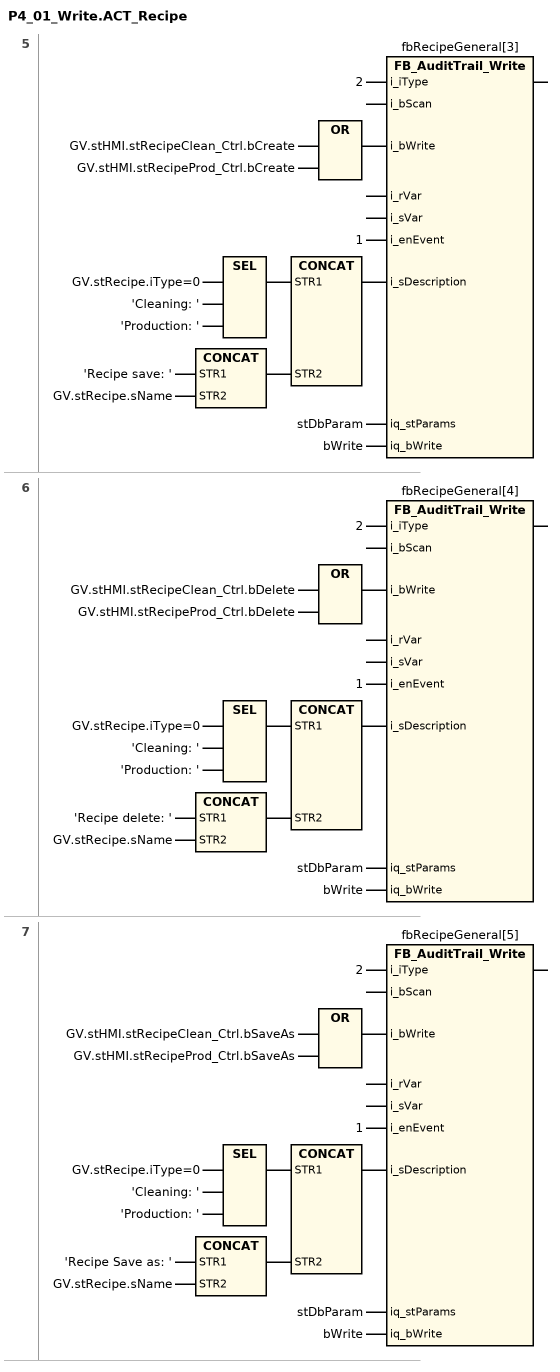
// NETWORK 5
fbRecipeGeneral[3](
    i_iType := 2,
    i_bWrite := GV.stHMI.stRecipeClean_Ctrl.bCreate OR GV.stHMI.stRecipeProd_Ctrl.bCreate,
    i_enEvent := 1,
    i_sDescription := CONCAT(STR1 := SEL(GV.stRecipe.iType=0, 'Cleaning: ', 'Production: '), STR2 := CONCAT(STR1 := 'Recipe save: ', STR2 := GV.stRecipe.sName)),
    iq_stParams := stDbParam,
    iq_bWrite := bWrite); // FB_AuditTrail_Write

// NETWORK 6
fbRecipeGeneral[4](
    i_iType := 2,
    i_bWrite := GV.stHMI.stRecipeClean_Ctrl.bDelete OR GV.stHMI.stRecipeProd_Ctrl.bDelete,
    i_enEvent := 1,
    i_sDescription := CONCAT(STR1 := SEL(GV.stRecipe.iType=0, 'Cleaning: ', 'Production: '), STR2 := CONCAT(STR1 := 'Recipe delete: ', STR2 := GV.stRecipe.sName)),
    iq_stParams := stDbParam,
    iq_bWrite := bWrite); // FB_AuditTrail_Write

// NETWORK 7
fbRecipeGeneral[5](
    i_iType := 2,
    i_bWrite := GV.stHMI.stRecipeClean_Ctrl.bSaveAs OR GV.stHMI.stRecipeProd_Ctrl.bSaveAs,
    i_enEvent := 1,
    i_sDescription := CONCAT(STR1 := SEL(GV.stRecipe.iType=0, 'Cleaning: ', 'Production: '), STR2 := CONCAT(STR1 := 'Recipe Save as: ', STR2 := GV.stRecipe.sName)),
    iq_stParams := stDbParam,
    iq_bWrite := bWrite); // FB_AuditTrail_Write

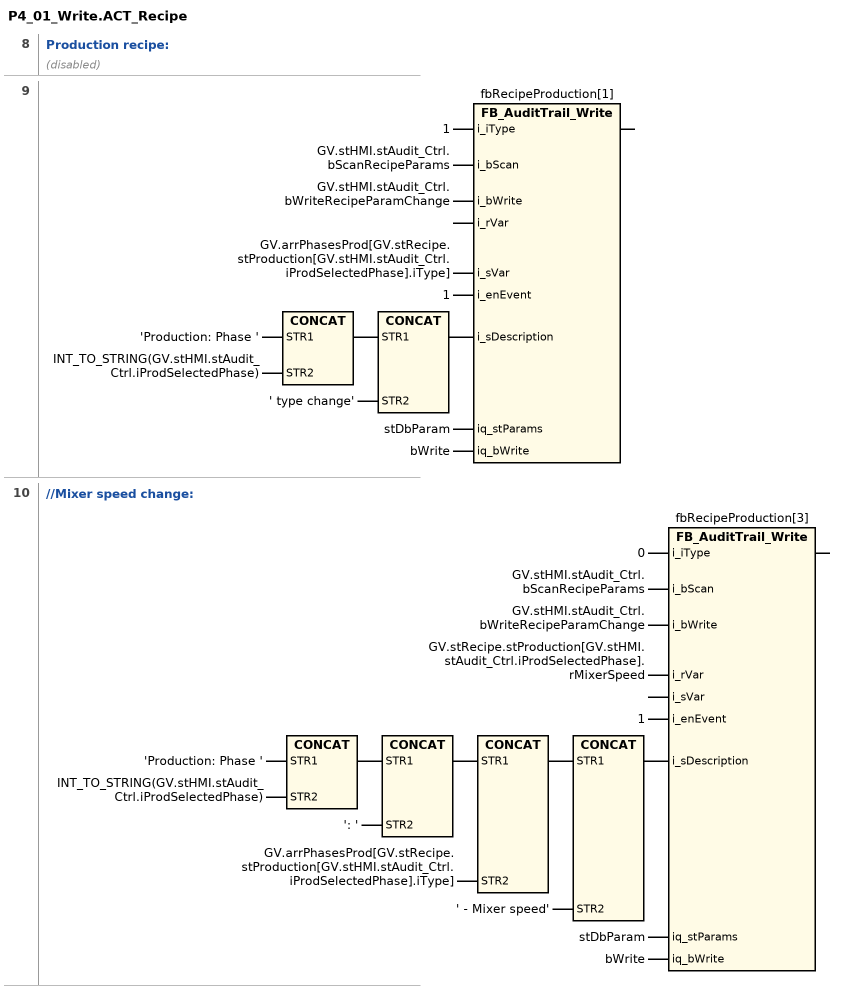
// NETWORK 8 (disabled)
// label: Production recipe

// NETWORK 9
fbRecipeProduction[1](
    i_iType := 1,
    i_bScan := GV.stHMI.stAudit_Ctrl.bScanRecipeParams,
    i_bWrite := GV.stHMI.stAudit_Ctrl.bWriteRecipeParamChange,
    i_sVar := GV.arrPhasesProd[GV.stRecipe.stProduction[GV.stHMI.stAudit_Ctrl.iProdSelectedPhase].iType],
    i_enEvent := 1,
    i_sDescription := CONCAT(STR1 := CONCAT(STR1 := 'Production: Phase ', STR2 := INT_TO_STRING(GV.stHMI.stAudit_Ctrl.iProdSelectedPhase)), STR2 := ' type change'),
    iq_stParams := stDbParam,
    iq_bWrite := bWrite); // FB_AuditTrail_Write

// NETWORK 10
// label: //Mixer speed change
fbRecipeProduction[3](
    i_iType := 0,
    i_bScan := GV.stHMI.stAudit_Ctrl.bScanRecipeParams,
    i_bWrite := GV.stHMI.stAudit_Ctrl.bWriteRecipeParamChange,
    i_rVar := GV.stRecipe.stProduction[GV.stHMI.stAudit_Ctrl.iProdSelectedPhase].rMixerSpeed,
    i_enEvent := 1,
    i_sDescription := CONCAT(STR1 := CONCAT(STR1 := CONCAT(STR1 := CONCAT(STR1 := 'Production: Phase ', STR2 := INT_TO_STRING(GV.stHMI.stAudit_Ctrl.iProdSelectedPhase)), STR2 := ': '), STR2 := GV.arrPhasesProd[GV.stRecipe.stProduction[GV.stHMI.stAudit_Ctrl.iProdSelectedPhase].iType]), STR2 := ' - Mixer speed'),
    iq_stParams := stDbParam,
    iq_bWrite := bWrite); // FB_AuditTrail_Write

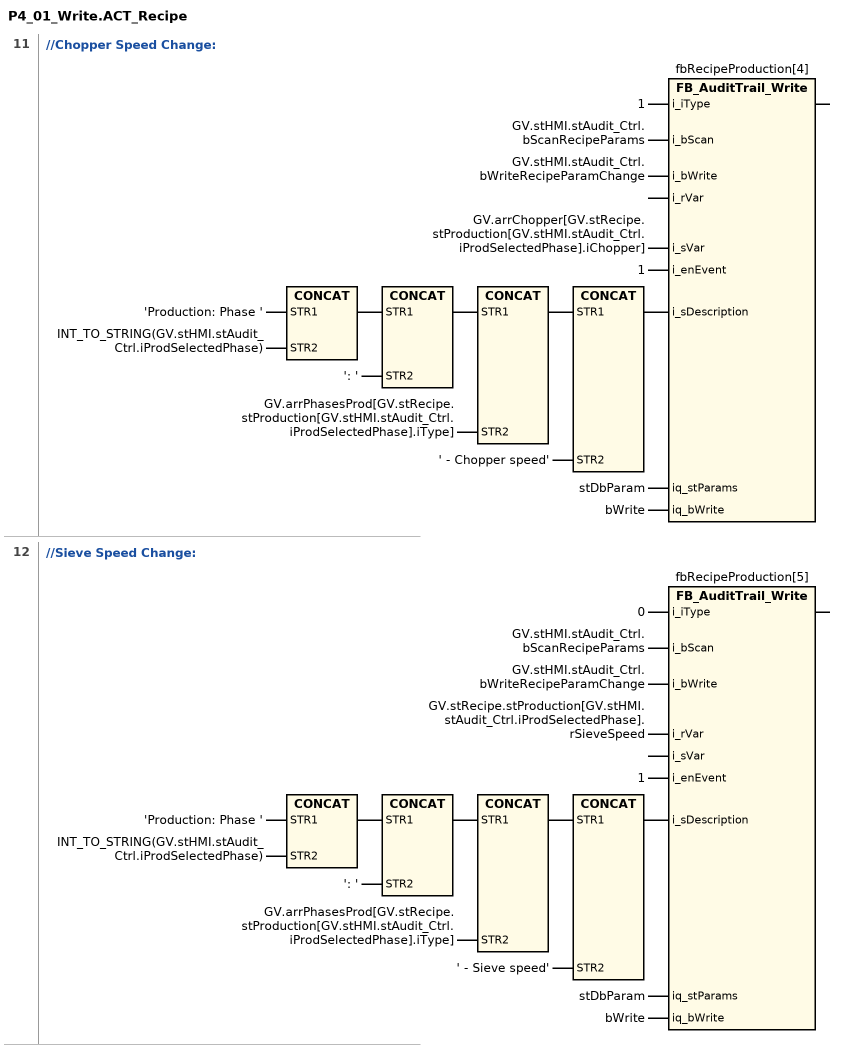
// NETWORK 11
// label: //Chopper Speed Change
fbRecipeProduction[4](
    i_iType := 1,
    i_bScan := GV.stHMI.stAudit_Ctrl.bScanRecipeParams,
    i_bWrite := GV.stHMI.stAudit_Ctrl.bWriteRecipeParamChange,
    i_sVar := GV.arrChopper[GV.stRecipe.stProduction[GV.stHMI.stAudit_Ctrl.iProdSelectedPhase].iChopper],
    i_enEvent := 1,
    i_sDescription := CONCAT(STR1 := CONCAT(STR1 := CONCAT(STR1 := CONCAT(STR1 := 'Production: Phase ', STR2 := INT_TO_STRING(GV.stHMI.stAudit_Ctrl.iProdSelectedPhase)), STR2 := ': '), STR2 := GV.arrPhasesProd[GV.stRecipe.stProduction[GV.stHMI.stAudit_Ctrl.iProdSelectedPhase].iType]), STR2 := ' - Chopper speed'),
    iq_stParams := stDbParam,
    iq_bWrite := bWrite); // FB_AuditTrail_Write

// NETWORK 12
// label: //Sieve Speed Change
fbRecipeProduction[5](
    i_iType := 0,
    i_bScan := GV.stHMI.stAudit_Ctrl.bScanRecipeParams,
    i_bWrite := GV.stHMI.stAudit_Ctrl.bWriteRecipeParamChange,
    i_rVar := GV.stRecipe.stProduction[GV.stHMI.stAudit_Ctrl.iProdSelectedPhase].rSieveSpeed,
    i_enEvent := 1,
    i_sDescription := CONCAT(STR1 := CONCAT(STR1 := CONCAT(STR1 := CONCAT(STR1 := 'Production: Phase ', STR2 := INT_TO_STRING(GV.stHMI.stAudit_Ctrl.iProdSelectedPhase)), STR2 := ': '), STR2 := GV.arrPhasesProd[GV.stRecipe.stProduction[GV.stHMI.stAudit_Ctrl.iProdSelectedPhase].iType]), STR2 := ' - Sieve speed'),
    iq_stParams := stDbParam,
    iq_bWrite := bWrite); // FB_AuditTrail_Write

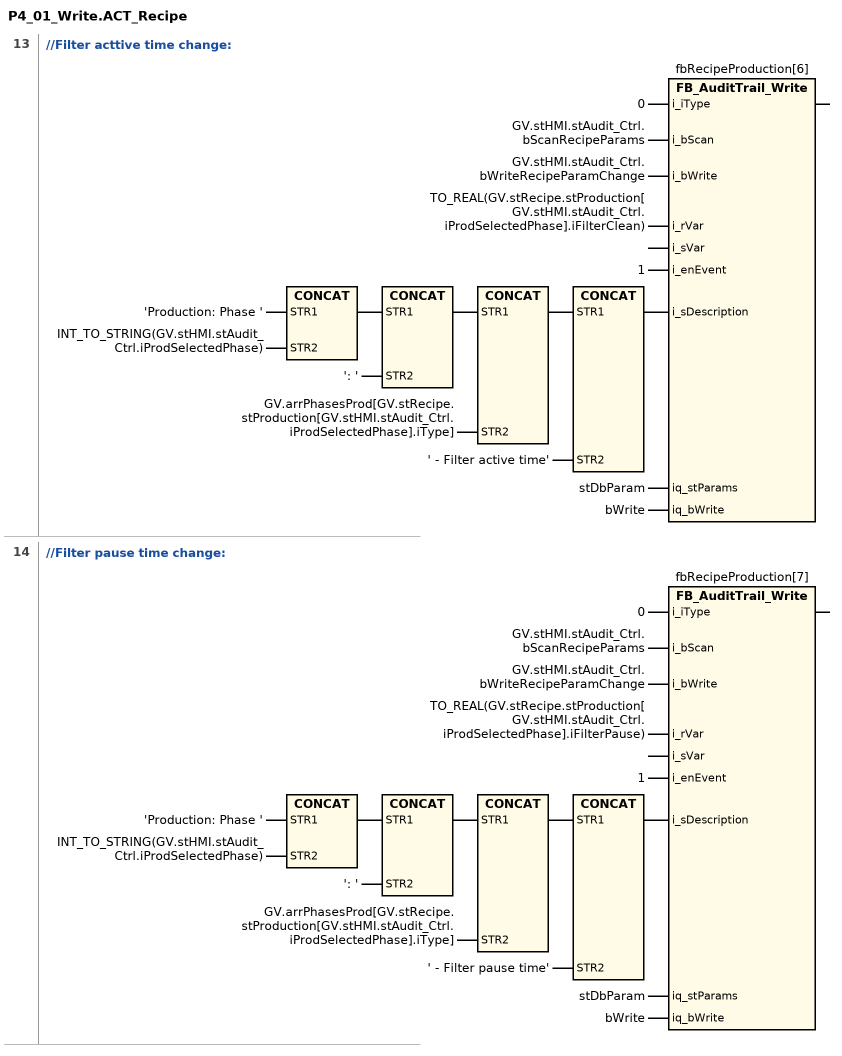
// NETWORK 13
// label: //Filter acttive time change
fbRecipeProduction[6](
    i_iType := 0,
    i_bScan := GV.stHMI.stAudit_Ctrl.bScanRecipeParams,
    i_bWrite := GV.stHMI.stAudit_Ctrl.bWriteRecipeParamChange,
    i_rVar := TO_REAL(GV.stRecipe.stProduction[GV.stHMI.stAudit_Ctrl.iProdSelectedPhase].iFilterClean),
    i_enEvent := 1,
    i_sDescription := CONCAT(STR1 := CONCAT(STR1 := CONCAT(STR1 := CONCAT(STR1 := 'Production: Phase ', STR2 := INT_TO_STRING(GV.stHMI.stAudit_Ctrl.iProdSelectedPhase)), STR2 := ': '), STR2 := GV.arrPhasesProd[GV.stRecipe.stProduction[GV.stHMI.stAudit_Ctrl.iProdSelectedPhase].iType]), STR2 := ' - Filter active time'),
    iq_stParams := stDbParam,
    iq_bWrite := bWrite); // FB_AuditTrail_Write

// NETWORK 14
// label: //Filter pause time change
fbRecipeProduction[7](
    i_iType := 0,
    i_bScan := GV.stHMI.stAudit_Ctrl.bScanRecipeParams,
    i_bWrite := GV.stHMI.stAudit_Ctrl.bWriteRecipeParamChange,
    i_rVar := TO_REAL(GV.stRecipe.stProduction[GV.stHMI.stAudit_Ctrl.iProdSelectedPhase].iFilterPause),
    i_enEvent := 1,
    i_sDescription := CONCAT(STR1 := CONCAT(STR1 := CONCAT(STR1 := CONCAT(STR1 := 'Production: Phase ', STR2 := INT_TO_STRING(GV.stHMI.stAudit_Ctrl.iProdSelectedPhase)), STR2 := ': '), STR2 := GV.arrPhasesProd[GV.stRecipe.stProduction[GV.stHMI.stAudit_Ctrl.iProdSelectedPhase].iType]), STR2 := ' - Filter pause time'),
    iq_stParams := stDbParam,
    iq_bWrite := bWrite); // FB_AuditTrail_Write

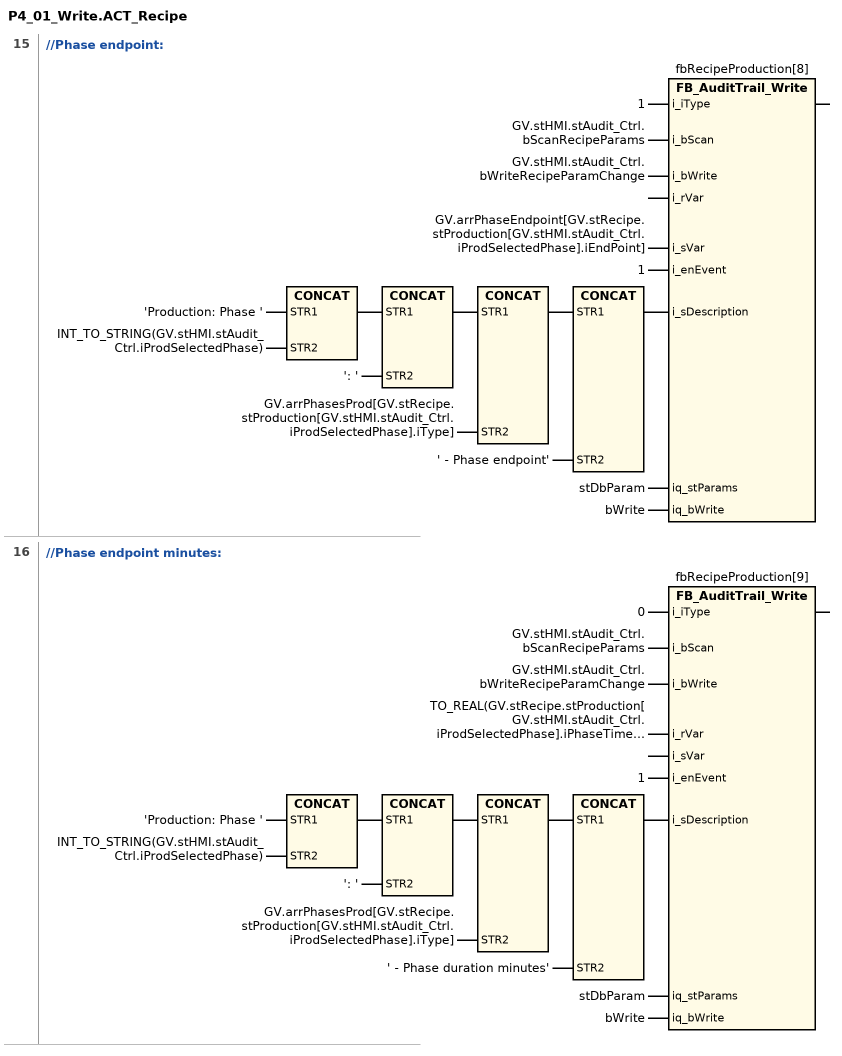
// NETWORK 15
// label: //Phase endpoint
fbRecipeProduction[8](
    i_iType := 1,
    i_bScan := GV.stHMI.stAudit_Ctrl.bScanRecipeParams,
    i_bWrite := GV.stHMI.stAudit_Ctrl.bWriteRecipeParamChange,
    i_sVar := GV.arrPhaseEndpoint[GV.stRecipe.stProduction[GV.stHMI.stAudit_Ctrl.iProdSelectedPhase].iEndPoint],
    i_enEvent := 1,
    i_sDescription := CONCAT(STR1 := CONCAT(STR1 := CONCAT(STR1 := CONCAT(STR1 := 'Production: Phase ', STR2 := INT_TO_STRING(GV.stHMI.stAudit_Ctrl.iProdSelectedPhase)), STR2 := ': '), STR2 := GV.arrPhasesProd[GV.stRecipe.stProduction[GV.stHMI.stAudit_Ctrl.iProdSelectedPhase].iType]), STR2 := ' - Phase endpoint'),
    iq_stParams := stDbParam,
    iq_bWrite := bWrite); // FB_AuditTrail_Write

// NETWORK 16
// label: //Phase endpoint minutes
fbRecipeProduction[9](
    i_iType := 0,
    i_bScan := GV.stHMI.stAudit_Ctrl.bScanRecipeParams,
    i_bWrite := GV.stHMI.stAudit_Ctrl.bWriteRecipeParamChange,
    i_rVar := TO_REAL(GV.stRecipe.stProduction[GV.stHMI.stAudit_Ctrl.iProdSelectedPhase].iPhaseTime.mins),
    i_enEvent := 1,
    i_sDescription := CONCAT(STR1 := CONCAT(STR1 := CONCAT(STR1 := CONCAT(STR1 := 'Production: Phase ', STR2 := INT_TO_STRING(GV.stHMI.stAudit_Ctrl.iProdSelectedPhase)), STR2 := ': '), STR2 := GV.arrPhasesProd[GV.stRecipe.stProduction[GV.stHMI.stAudit_Ctrl.iProdSelectedPhase].iType]), STR2 := ' - Phase duration minutes'),
    iq_stParams := stDbParam,
    iq_bWrite := bWrite); // FB_AuditTrail_Write

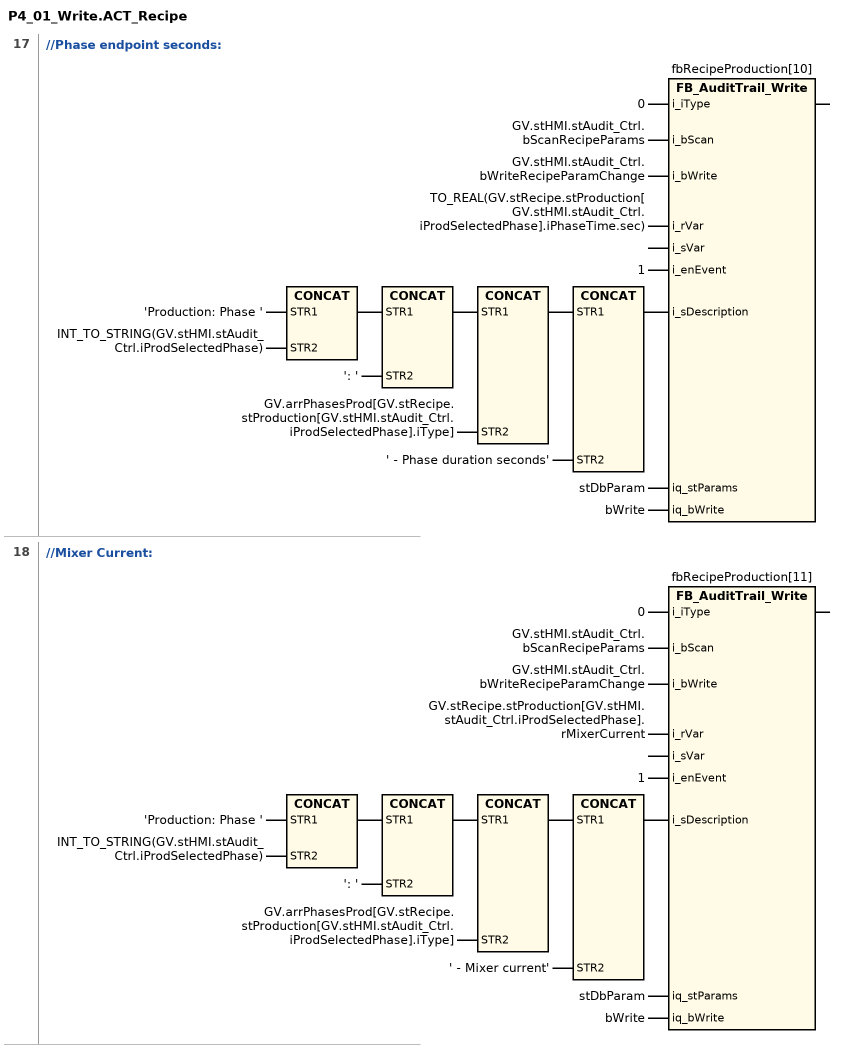
// NETWORK 17
// label: //Phase endpoint seconds
fbRecipeProduction[10](
    i_iType := 0,
    i_bScan := GV.stHMI.stAudit_Ctrl.bScanRecipeParams,
    i_bWrite := GV.stHMI.stAudit_Ctrl.bWriteRecipeParamChange,
    i_rVar := TO_REAL(GV.stRecipe.stProduction[GV.stHMI.stAudit_Ctrl.iProdSelectedPhase].iPhaseTime.sec),
    i_enEvent := 1,
    i_sDescription := CONCAT(STR1 := CONCAT(STR1 := CONCAT(STR1 := CONCAT(STR1 := 'Production: Phase ', STR2 := INT_TO_STRING(GV.stHMI.stAudit_Ctrl.iProdSelectedPhase)), STR2 := ': '), STR2 := GV.arrPhasesProd[GV.stRecipe.stProduction[GV.stHMI.stAudit_Ctrl.iProdSelectedPhase].iType]), STR2 := ' - Phase duration seconds'),
    iq_stParams := stDbParam,
    iq_bWrite := bWrite); // FB_AuditTrail_Write

// NETWORK 18
// label: //Mixer Current
fbRecipeProduction[11](
    i_iType := 0,
    i_bScan := GV.stHMI.stAudit_Ctrl.bScanRecipeParams,
    i_bWrite := GV.stHMI.stAudit_Ctrl.bWriteRecipeParamChange,
    i_rVar := GV.stRecipe.stProduction[GV.stHMI.stAudit_Ctrl.iProdSelectedPhase].rMixerCurrent,
    i_enEvent := 1,
    i_sDescription := CONCAT(STR1 := CONCAT(STR1 := CONCAT(STR1 := CONCAT(STR1 := 'Production: Phase ', STR2 := INT_TO_STRING(GV.stHMI.stAudit_Ctrl.iProdSelectedPhase)), STR2 := ': '), STR2 := GV.arrPhasesProd[GV.stRecipe.stProduction[GV.stHMI.stAudit_Ctrl.iProdSelectedPhase].iType]), STR2 := ' - Mixer current'),
    iq_stParams := stDbParam,
    iq_bWrite := bWrite); // FB_AuditTrail_Write

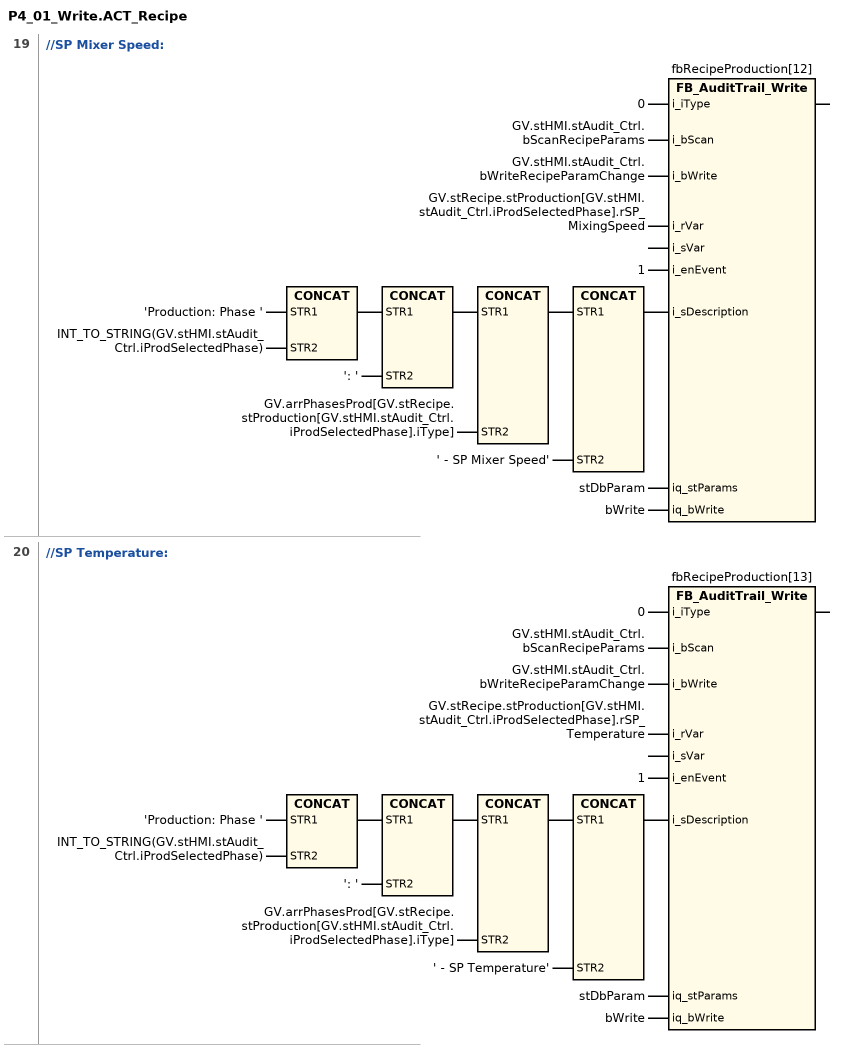
// NETWORK 19
// label: //SP Mixer Speed
fbRecipeProduction[12](
    i_iType := 0,
    i_bScan := GV.stHMI.stAudit_Ctrl.bScanRecipeParams,
    i_bWrite := GV.stHMI.stAudit_Ctrl.bWriteRecipeParamChange,
    i_rVar := GV.stRecipe.stProduction[GV.stHMI.stAudit_Ctrl.iProdSelectedPhase].rSP_MixingSpeed,
    i_enEvent := 1,
    i_sDescription := CONCAT(STR1 := CONCAT(STR1 := CONCAT(STR1 := CONCAT(STR1 := 'Production: Phase ', STR2 := INT_TO_STRING(GV.stHMI.stAudit_Ctrl.iProdSelectedPhase)), STR2 := ': '), STR2 := GV.arrPhasesProd[GV.stRecipe.stProduction[GV.stHMI.stAudit_Ctrl.iProdSelectedPhase].iType]), STR2 := ' - SP Mixer Speed'),
    iq_stParams := stDbParam,
    iq_bWrite := bWrite); // FB_AuditTrail_Write

// NETWORK 20
// label: //SP Temperature
fbRecipeProduction[13](
    i_iType := 0,
    i_bScan := GV.stHMI.stAudit_Ctrl.bScanRecipeParams,
    i_bWrite := GV.stHMI.stAudit_Ctrl.bWriteRecipeParamChange,
    i_rVar := GV.stRecipe.stProduction[GV.stHMI.stAudit_Ctrl.iProdSelectedPhase].rSP_Temperature,
    i_enEvent := 1,
    i_sDescription := CONCAT(STR1 := CONCAT(STR1 := CONCAT(STR1 := CONCAT(STR1 := 'Production: Phase ', STR2 := INT_TO_STRING(GV.stHMI.stAudit_Ctrl.iProdSelectedPhase)), STR2 := ': '), STR2 := GV.arrPhasesProd[GV.stRecipe.stProduction[GV.stHMI.stAudit_Ctrl.iProdSelectedPhase].iType]), STR2 := ' - SP Temperature'),
    iq_stParams := stDbParam,
    iq_bWrite := bWrite); // FB_AuditTrail_Write

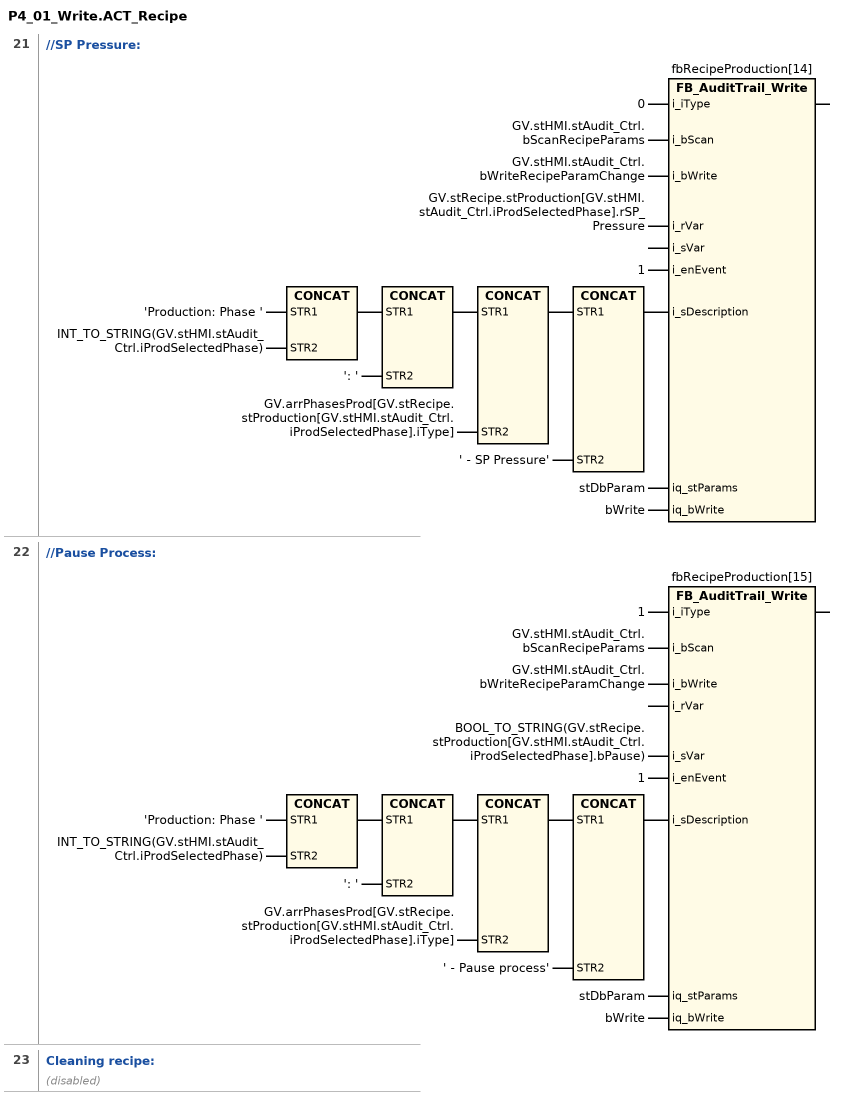
// NETWORK 21
// label: //SP Pressure
fbRecipeProduction[14](
    i_iType := 0,
    i_bScan := GV.stHMI.stAudit_Ctrl.bScanRecipeParams,
    i_bWrite := GV.stHMI.stAudit_Ctrl.bWriteRecipeParamChange,
    i_rVar := GV.stRecipe.stProduction[GV.stHMI.stAudit_Ctrl.iProdSelectedPhase].rSP_Pressure,
    i_enEvent := 1,
    i_sDescription := CONCAT(STR1 := CONCAT(STR1 := CONCAT(STR1 := CONCAT(STR1 := 'Production: Phase ', STR2 := INT_TO_STRING(GV.stHMI.stAudit_Ctrl.iProdSelectedPhase)), STR2 := ': '), STR2 := GV.arrPhasesProd[GV.stRecipe.stProduction[GV.stHMI.stAudit_Ctrl.iProdSelectedPhase].iType]), STR2 := ' - SP Pressure'),
    iq_stParams := stDbParam,
    iq_bWrite := bWrite); // FB_AuditTrail_Write

// NETWORK 22
// label: //Pause Process
fbRecipeProduction[15](
    i_iType := 1,
    i_bScan := GV.stHMI.stAudit_Ctrl.bScanRecipeParams,
    i_bWrite := GV.stHMI.stAudit_Ctrl.bWriteRecipeParamChange,
    i_sVar := BOOL_TO_STRING(GV.stRecipe.stProduction[GV.stHMI.stAudit_Ctrl.iProdSelectedPhase].bPause),
    i_enEvent := 1,
    i_sDescription := CONCAT(STR1 := CONCAT(STR1 := CONCAT(STR1 := CONCAT(STR1 := 'Production: Phase ', STR2 := INT_TO_STRING(GV.stHMI.stAudit_Ctrl.iProdSelectedPhase)), STR2 := ': '), STR2 := GV.arrPhasesProd[GV.stRecipe.stProduction[GV.stHMI.stAudit_Ctrl.iProdSelectedPhase].iType]), STR2 := ' - Pause process'),
    iq_stParams := stDbParam,
    iq_bWrite := bWrite); // FB_AuditTrail_Write

// NETWORK 23 (disabled)
// label: Cleaning recipe

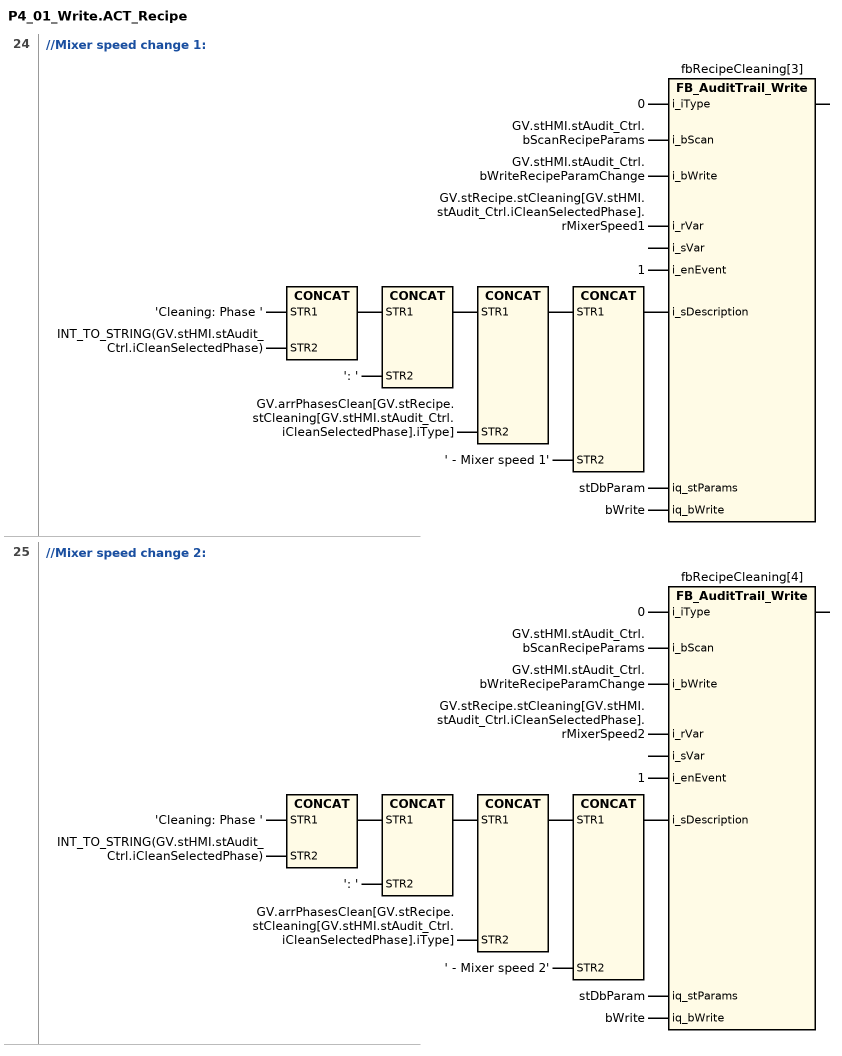
// NETWORK 24
// label: //Mixer speed change 1
fbRecipeCleaning[3](
    i_iType := 0,
    i_bScan := GV.stHMI.stAudit_Ctrl.bScanRecipeParams,
    i_bWrite := GV.stHMI.stAudit_Ctrl.bWriteRecipeParamChange,
    i_rVar := GV.stRecipe.stCleaning[GV.stHMI.stAudit_Ctrl.iCleanSelectedPhase].rMixerSpeed1,
    i_enEvent := 1,
    i_sDescription := CONCAT(STR1 := CONCAT(STR1 := CONCAT(STR1 := CONCAT(STR1 := 'Cleaning: Phase ', STR2 := INT_TO_STRING(GV.stHMI.stAudit_Ctrl.iCleanSelectedPhase)), STR2 := ': '), STR2 := GV.arrPhasesClean[GV.stRecipe.stCleaning[GV.stHMI.stAudit_Ctrl.iCleanSelectedPhase].iType]), STR2 := ' - Mixer speed 1'),
    iq_stParams := stDbParam,
    iq_bWrite := bWrite); // FB_AuditTrail_Write

// NETWORK 25
// label: //Mixer speed change 2
fbRecipeCleaning[4](
    i_iType := 0,
    i_bScan := GV.stHMI.stAudit_Ctrl.bScanRecipeParams,
    i_bWrite := GV.stHMI.stAudit_Ctrl.bWriteRecipeParamChange,
    i_rVar := GV.stRecipe.stCleaning[GV.stHMI.stAudit_Ctrl.iCleanSelectedPhase].rMixerSpeed2,
    i_enEvent := 1,
    i_sDescription := CONCAT(STR1 := CONCAT(STR1 := CONCAT(STR1 := CONCAT(STR1 := 'Cleaning: Phase ', STR2 := INT_TO_STRING(GV.stHMI.stAudit_Ctrl.iCleanSelectedPhase)), STR2 := ': '), STR2 := GV.arrPhasesClean[GV.stRecipe.stCleaning[GV.stHMI.stAudit_Ctrl.iCleanSelectedPhase].iType]), STR2 := ' - Mixer speed 2'),
    iq_stParams := stDbParam,
    iq_bWrite := bWrite); // FB_AuditTrail_Write

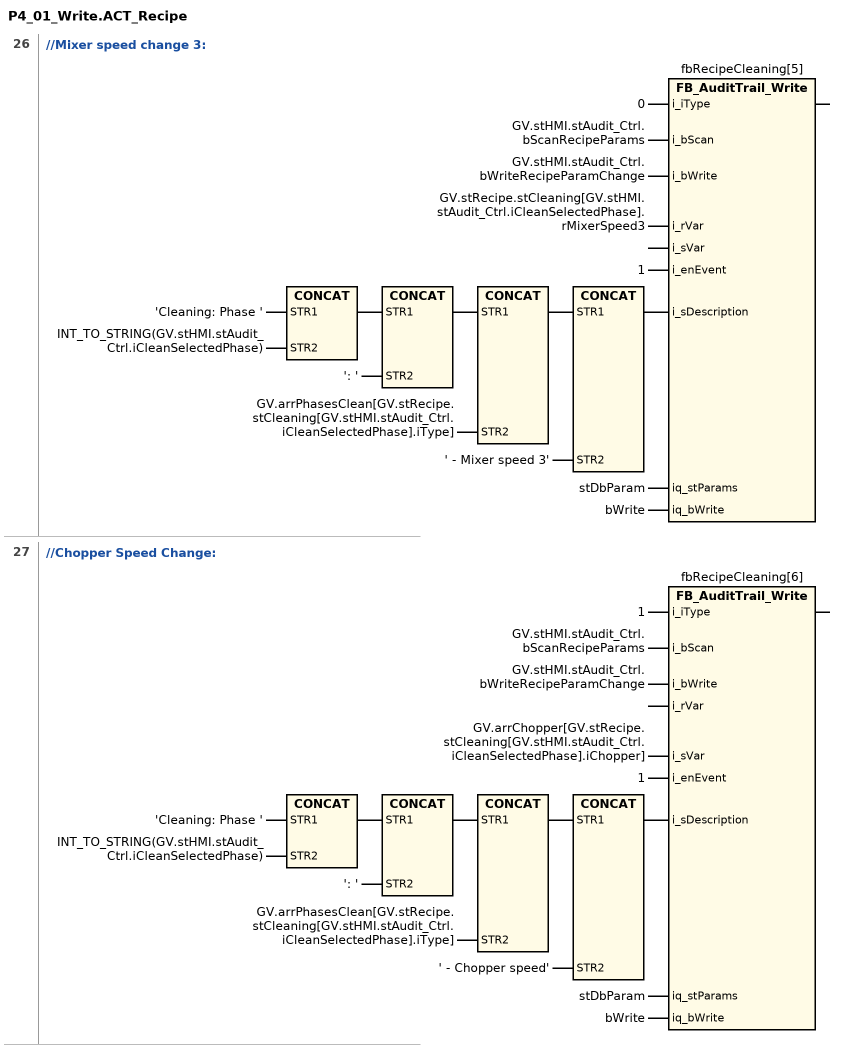
// NETWORK 26
// label: //Mixer speed change 3
fbRecipeCleaning[5](
    i_iType := 0,
    i_bScan := GV.stHMI.stAudit_Ctrl.bScanRecipeParams,
    i_bWrite := GV.stHMI.stAudit_Ctrl.bWriteRecipeParamChange,
    i_rVar := GV.stRecipe.stCleaning[GV.stHMI.stAudit_Ctrl.iCleanSelectedPhase].rMixerSpeed3,
    i_enEvent := 1,
    i_sDescription := CONCAT(STR1 := CONCAT(STR1 := CONCAT(STR1 := CONCAT(STR1 := 'Cleaning: Phase ', STR2 := INT_TO_STRING(GV.stHMI.stAudit_Ctrl.iCleanSelectedPhase)), STR2 := ': '), STR2 := GV.arrPhasesClean[GV.stRecipe.stCleaning[GV.stHMI.stAudit_Ctrl.iCleanSelectedPhase].iType]), STR2 := ' - Mixer speed 3'),
    iq_stParams := stDbParam,
    iq_bWrite := bWrite); // FB_AuditTrail_Write

// NETWORK 27
// label: //Chopper Speed Change
fbRecipeCleaning[6](
    i_iType := 1,
    i_bScan := GV.stHMI.stAudit_Ctrl.bScanRecipeParams,
    i_bWrite := GV.stHMI.stAudit_Ctrl.bWriteRecipeParamChange,
    i_sVar := GV.arrChopper[GV.stRecipe.stCleaning[GV.stHMI.stAudit_Ctrl.iCleanSelectedPhase].iChopper],
    i_enEvent := 1,
    i_sDescription := CONCAT(STR1 := CONCAT(STR1 := CONCAT(STR1 := CONCAT(STR1 := 'Cleaning: Phase ', STR2 := INT_TO_STRING(GV.stHMI.stAudit_Ctrl.iCleanSelectedPhase)), STR2 := ': '), STR2 := GV.arrPhasesClean[GV.stRecipe.stCleaning[GV.stHMI.stAudit_Ctrl.iCleanSelectedPhase].iType]), STR2 := ' - Chopper speed'),
    iq_stParams := stDbParam,
    iq_bWrite := bWrite); // FB_AuditTrail_Write

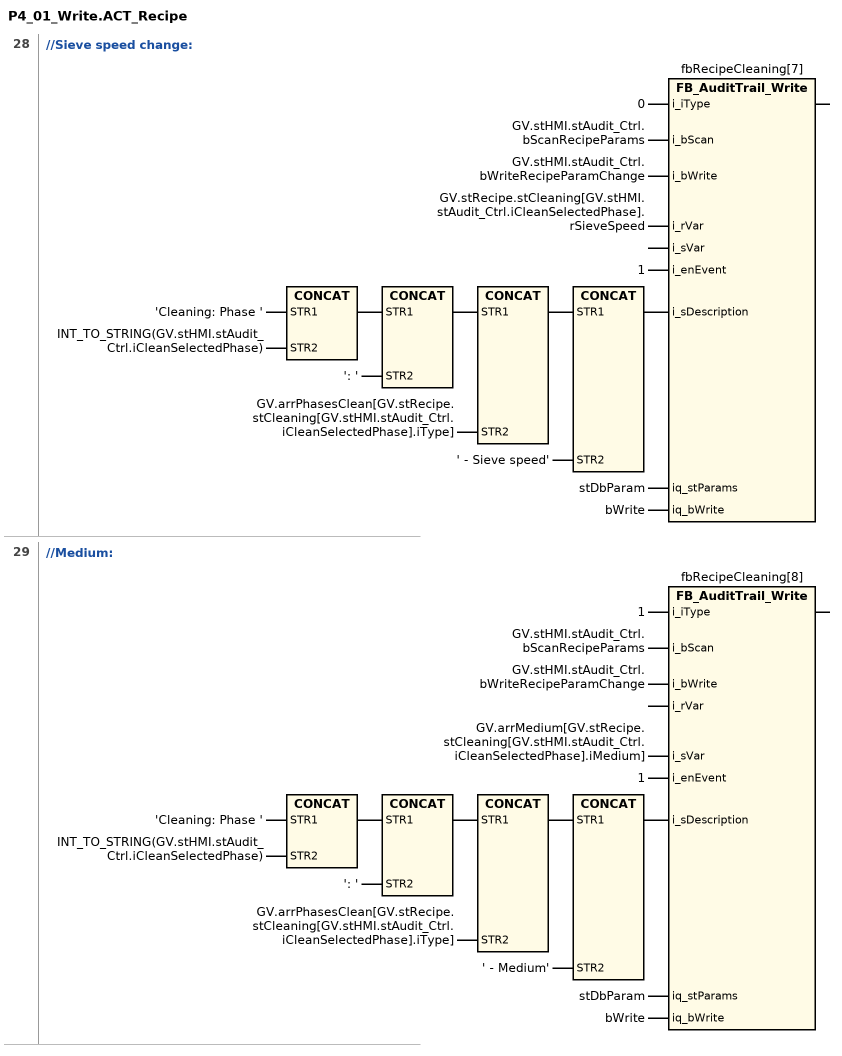
// NETWORK 28
// label: //Sieve speed change
fbRecipeCleaning[7](
    i_iType := 0,
    i_bScan := GV.stHMI.stAudit_Ctrl.bScanRecipeParams,
    i_bWrite := GV.stHMI.stAudit_Ctrl.bWriteRecipeParamChange,
    i_rVar := GV.stRecipe.stCleaning[GV.stHMI.stAudit_Ctrl.iCleanSelectedPhase].rSieveSpeed,
    i_enEvent := 1,
    i_sDescription := CONCAT(STR1 := CONCAT(STR1 := CONCAT(STR1 := CONCAT(STR1 := 'Cleaning: Phase ', STR2 := INT_TO_STRING(GV.stHMI.stAudit_Ctrl.iCleanSelectedPhase)), STR2 := ': '), STR2 := GV.arrPhasesClean[GV.stRecipe.stCleaning[GV.stHMI.stAudit_Ctrl.iCleanSelectedPhase].iType]), STR2 := ' - Sieve speed'),
    iq_stParams := stDbParam,
    iq_bWrite := bWrite); // FB_AuditTrail_Write

// NETWORK 29
// label: //Medium
fbRecipeCleaning[8](
    i_iType := 1,
    i_bScan := GV.stHMI.stAudit_Ctrl.bScanRecipeParams,
    i_bWrite := GV.stHMI.stAudit_Ctrl.bWriteRecipeParamChange,
    i_sVar := GV.arrMedium[GV.stRecipe.stCleaning[GV.stHMI.stAudit_Ctrl.iCleanSelectedPhase].iMedium],
    i_enEvent := 1,
    i_sDescription := CONCAT(STR1 := CONCAT(STR1 := CONCAT(STR1 := CONCAT(STR1 := 'Cleaning: Phase ', STR2 := INT_TO_STRING(GV.stHMI.stAudit_Ctrl.iCleanSelectedPhase)), STR2 := ': '), STR2 := GV.arrPhasesClean[GV.stRecipe.stCleaning[GV.stHMI.stAudit_Ctrl.iCleanSelectedPhase].iType]), STR2 := ' - Medium'),
    iq_stParams := stDbParam,
    iq_bWrite := bWrite); // FB_AuditTrail_Write

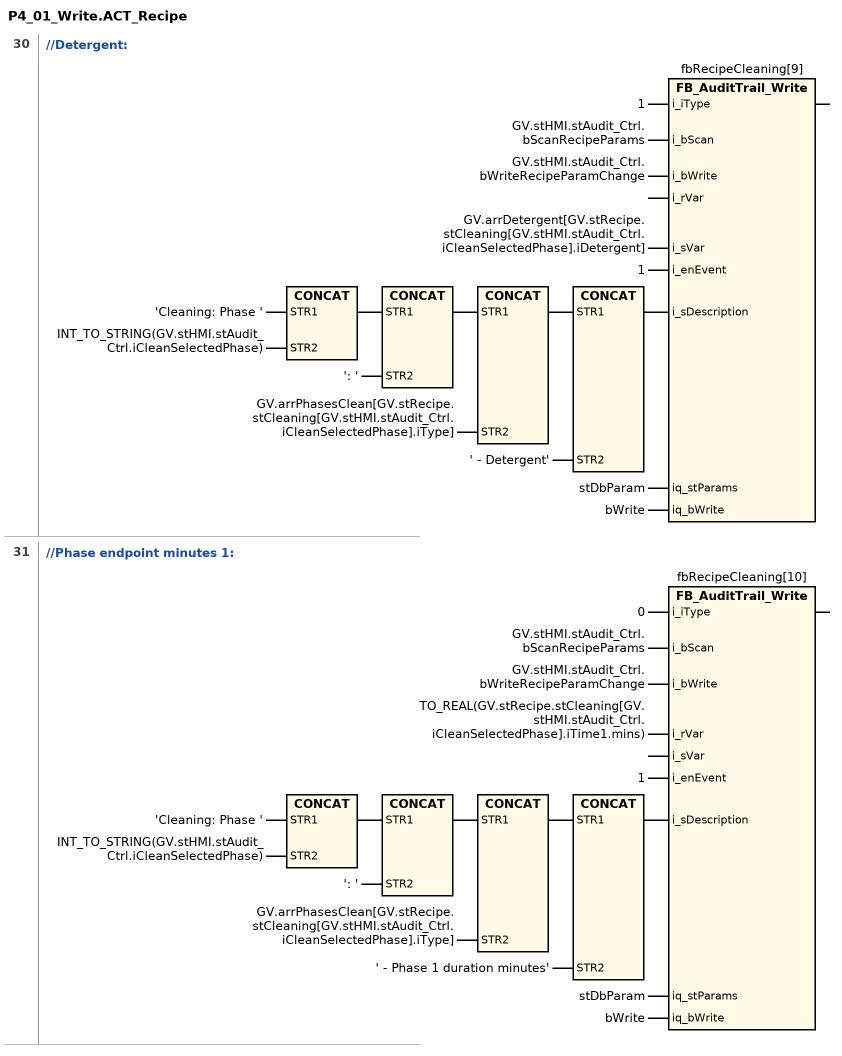
// NETWORK 30
// label: //Detergent
fbRecipeCleaning[9](
    i_iType := 1,
    i_bScan := GV.stHMI.stAudit_Ctrl.bScanRecipeParams,
    i_bWrite := GV.stHMI.stAudit_Ctrl.bWriteRecipeParamChange,
    i_sVar := GV.arrDetergent[GV.stRecipe.stCleaning[GV.stHMI.stAudit_Ctrl.iCleanSelectedPhase].iDetergent],
    i_enEvent := 1,
    i_sDescription := CONCAT(STR1 := CONCAT(STR1 := CONCAT(STR1 := CONCAT(STR1 := 'Cleaning: Phase ', STR2 := INT_TO_STRING(GV.stHMI.stAudit_Ctrl.iCleanSelectedPhase)), STR2 := ': '), STR2 := GV.arrPhasesClean[GV.stRecipe.stCleaning[GV.stHMI.stAudit_Ctrl.iCleanSelectedPhase].iType]), STR2 := ' - Detergent'),
    iq_stParams := stDbParam,
    iq_bWrite := bWrite); // FB_AuditTrail_Write

// NETWORK 31
// label: //Phase endpoint minutes 1
fbRecipeCleaning[10](
    i_iType := 0,
    i_bScan := GV.stHMI.stAudit_Ctrl.bScanRecipeParams,
    i_bWrite := GV.stHMI.stAudit_Ctrl.bWriteRecipeParamChange,
    i_rVar := TO_REAL(GV.stRecipe.stCleaning[GV.stHMI.stAudit_Ctrl.iCleanSelectedPhase].iTime1.mins),
    i_enEvent := 1,
    i_sDescription := CONCAT(STR1 := CONCAT(STR1 := CONCAT(STR1 := CONCAT(STR1 := 'Cleaning: Phase ', STR2 := INT_TO_STRING(GV.stHMI.stAudit_Ctrl.iCleanSelectedPhase)), STR2 := ': '), STR2 := GV.arrPhasesClean[GV.stRecipe.stCleaning[GV.stHMI.stAudit_Ctrl.iCleanSelectedPhase].iType]), STR2 := ' - Phase 1 duration minutes'),
    iq_stParams := stDbParam,
    iq_bWrite := bWrite); // FB_AuditTrail_Write

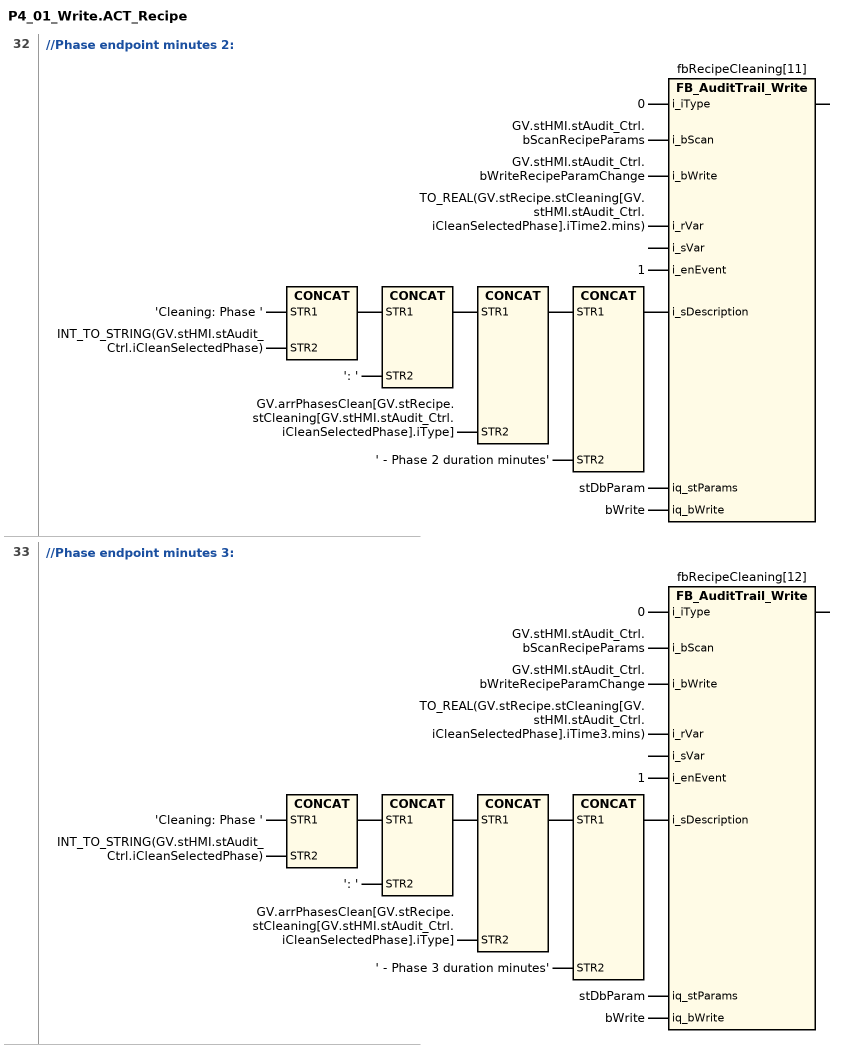
// NETWORK 32
// label: //Phase endpoint minutes 2
fbRecipeCleaning[11](
    i_iType := 0,
    i_bScan := GV.stHMI.stAudit_Ctrl.bScanRecipeParams,
    i_bWrite := GV.stHMI.stAudit_Ctrl.bWriteRecipeParamChange,
    i_rVar := TO_REAL(GV.stRecipe.stCleaning[GV.stHMI.stAudit_Ctrl.iCleanSelectedPhase].iTime2.mins),
    i_enEvent := 1,
    i_sDescription := CONCAT(STR1 := CONCAT(STR1 := CONCAT(STR1 := CONCAT(STR1 := 'Cleaning: Phase ', STR2 := INT_TO_STRING(GV.stHMI.stAudit_Ctrl.iCleanSelectedPhase)), STR2 := ': '), STR2 := GV.arrPhasesClean[GV.stRecipe.stCleaning[GV.stHMI.stAudit_Ctrl.iCleanSelectedPhase].iType]), STR2 := ' - Phase 2 duration minutes'),
    iq_stParams := stDbParam,
    iq_bWrite := bWrite); // FB_AuditTrail_Write

// NETWORK 33
// label: //Phase endpoint minutes 3
fbRecipeCleaning[12](
    i_iType := 0,
    i_bScan := GV.stHMI.stAudit_Ctrl.bScanRecipeParams,
    i_bWrite := GV.stHMI.stAudit_Ctrl.bWriteRecipeParamChange,
    i_rVar := TO_REAL(GV.stRecipe.stCleaning[GV.stHMI.stAudit_Ctrl.iCleanSelectedPhase].iTime3.mins),
    i_enEvent := 1,
    i_sDescription := CONCAT(STR1 := CONCAT(STR1 := CONCAT(STR1 := CONCAT(STR1 := 'Cleaning: Phase ', STR2 := INT_TO_STRING(GV.stHMI.stAudit_Ctrl.iCleanSelectedPhase)), STR2 := ': '), STR2 := GV.arrPhasesClean[GV.stRecipe.stCleaning[GV.stHMI.stAudit_Ctrl.iCleanSelectedPhase].iType]), STR2 := ' - Phase 3 duration minutes'),
    iq_stParams := stDbParam,
    iq_bWrite := bWrite); // FB_AuditTrail_Write

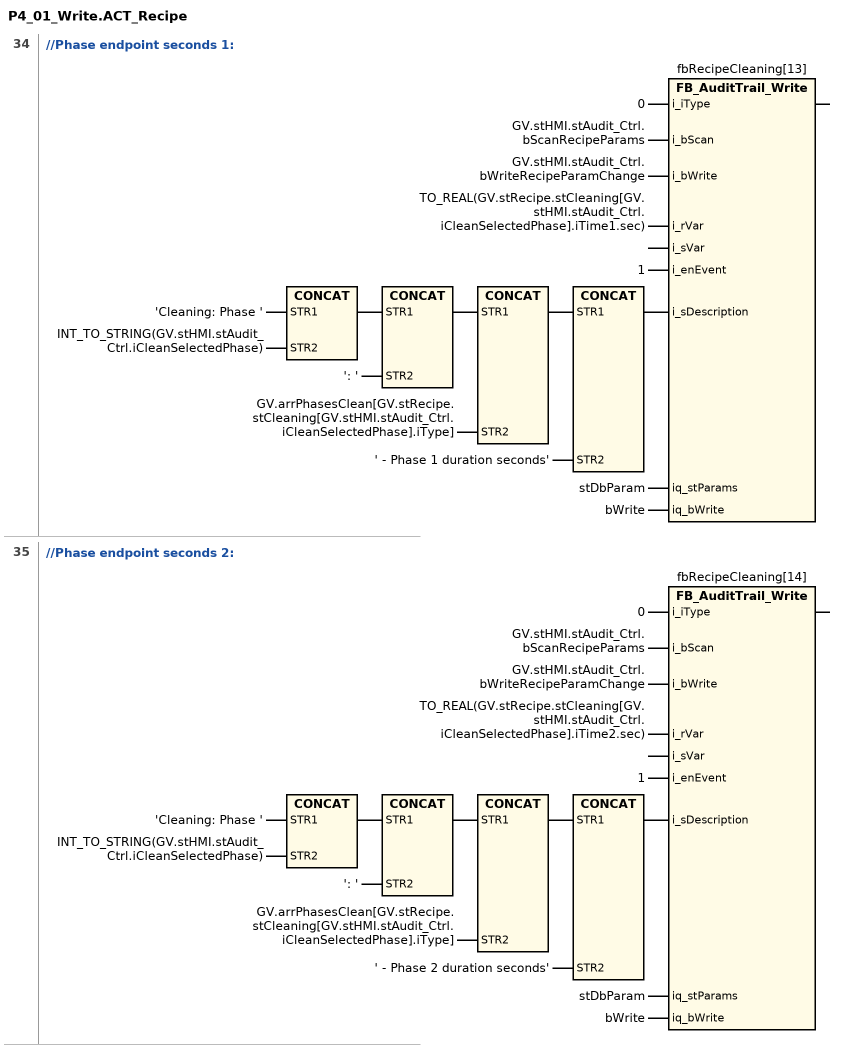
// NETWORK 34
// label: //Phase endpoint seconds 1
fbRecipeCleaning[13](
    i_iType := 0,
    i_bScan := GV.stHMI.stAudit_Ctrl.bScanRecipeParams,
    i_bWrite := GV.stHMI.stAudit_Ctrl.bWriteRecipeParamChange,
    i_rVar := TO_REAL(GV.stRecipe.stCleaning[GV.stHMI.stAudit_Ctrl.iCleanSelectedPhase].iTime1.sec),
    i_enEvent := 1,
    i_sDescription := CONCAT(STR1 := CONCAT(STR1 := CONCAT(STR1 := CONCAT(STR1 := 'Cleaning: Phase ', STR2 := INT_TO_STRING(GV.stHMI.stAudit_Ctrl.iCleanSelectedPhase)), STR2 := ': '), STR2 := GV.arrPhasesClean[GV.stRecipe.stCleaning[GV.stHMI.stAudit_Ctrl.iCleanSelectedPhase].iType]), STR2 := ' - Phase 1 duration seconds'),
    iq_stParams := stDbParam,
    iq_bWrite := bWrite); // FB_AuditTrail_Write

// NETWORK 35
// label: //Phase endpoint seconds 2
fbRecipeCleaning[14](
    i_iType := 0,
    i_bScan := GV.stHMI.stAudit_Ctrl.bScanRecipeParams,
    i_bWrite := GV.stHMI.stAudit_Ctrl.bWriteRecipeParamChange,
    i_rVar := TO_REAL(GV.stRecipe.stCleaning[GV.stHMI.stAudit_Ctrl.iCleanSelectedPhase].iTime2.sec),
    i_enEvent := 1,
    i_sDescription := CONCAT(STR1 := CONCAT(STR1 := CONCAT(STR1 := CONCAT(STR1 := 'Cleaning: Phase ', STR2 := INT_TO_STRING(GV.stHMI.stAudit_Ctrl.iCleanSelectedPhase)), STR2 := ': '), STR2 := GV.arrPhasesClean[GV.stRecipe.stCleaning[GV.stHMI.stAudit_Ctrl.iCleanSelectedPhase].iType]), STR2 := ' - Phase 2 duration seconds'),
    iq_stParams := stDbParam,
    iq_bWrite := bWrite); // FB_AuditTrail_Write

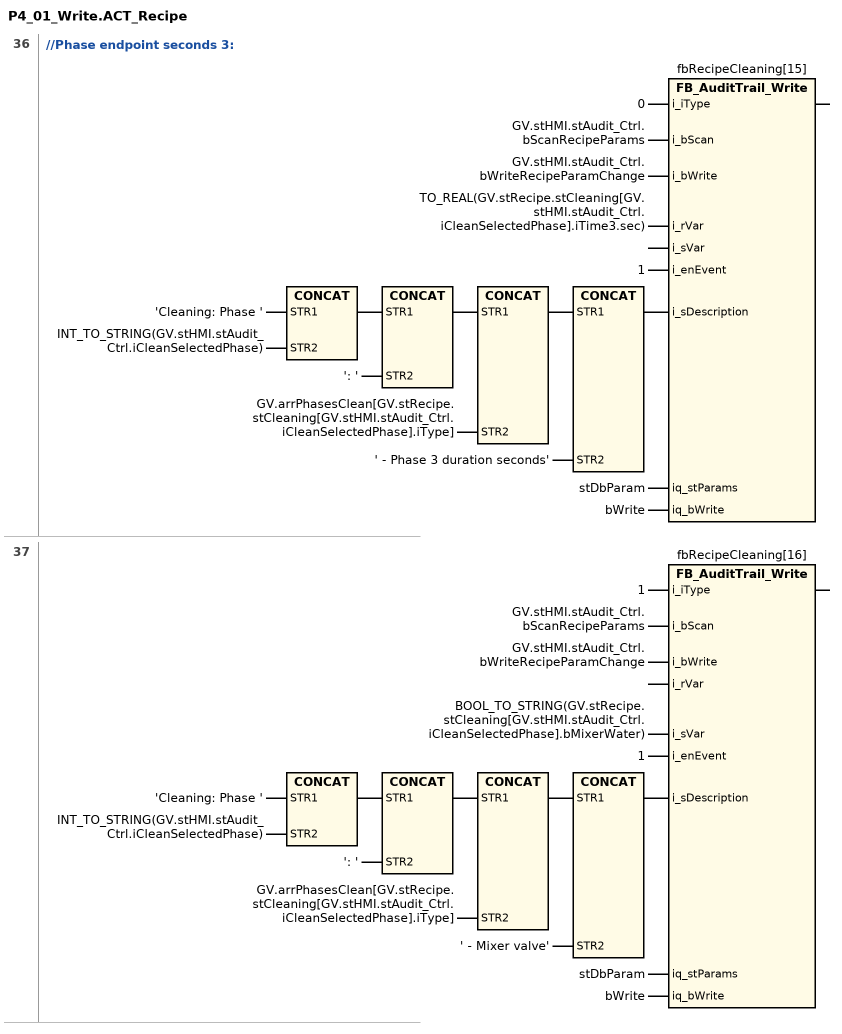
// NETWORK 36
// label: //Phase endpoint seconds 3
fbRecipeCleaning[15](
    i_iType := 0,
    i_bScan := GV.stHMI.stAudit_Ctrl.bScanRecipeParams,
    i_bWrite := GV.stHMI.stAudit_Ctrl.bWriteRecipeParamChange,
    i_rVar := TO_REAL(GV.stRecipe.stCleaning[GV.stHMI.stAudit_Ctrl.iCleanSelectedPhase].iTime3.sec),
    i_enEvent := 1,
    i_sDescription := CONCAT(STR1 := CONCAT(STR1 := CONCAT(STR1 := CONCAT(STR1 := 'Cleaning: Phase ', STR2 := INT_TO_STRING(GV.stHMI.stAudit_Ctrl.iCleanSelectedPhase)), STR2 := ': '), STR2 := GV.arrPhasesClean[GV.stRecipe.stCleaning[GV.stHMI.stAudit_Ctrl.iCleanSelectedPhase].iType]), STR2 := ' - Phase 3 duration seconds'),
    iq_stParams := stDbParam,
    iq_bWrite := bWrite); // FB_AuditTrail_Write

// NETWORK 37
fbRecipeCleaning[16](
    i_iType := 1,
    i_bScan := GV.stHMI.stAudit_Ctrl.bScanRecipeParams,
    i_bWrite := GV.stHMI.stAudit_Ctrl.bWriteRecipeParamChange,
    i_sVar := BOOL_TO_STRING(GV.stRecipe.stCleaning[GV.stHMI.stAudit_Ctrl.iCleanSelectedPhase].bMixerWater),
    i_enEvent := 1,
    i_sDescription := CONCAT(STR1 := CONCAT(STR1 := CONCAT(STR1 := CONCAT(STR1 := 'Cleaning: Phase ', STR2 := INT_TO_STRING(GV.stHMI.stAudit_Ctrl.iCleanSelectedPhase)), STR2 := ': '), STR2 := GV.arrPhasesClean[GV.stRecipe.stCleaning[GV.stHMI.stAudit_Ctrl.iCleanSelectedPhase].iType]), STR2 := ' - Mixer valve'),
    iq_stParams := stDbParam,
    iq_bWrite := bWrite); // FB_AuditTrail_Write

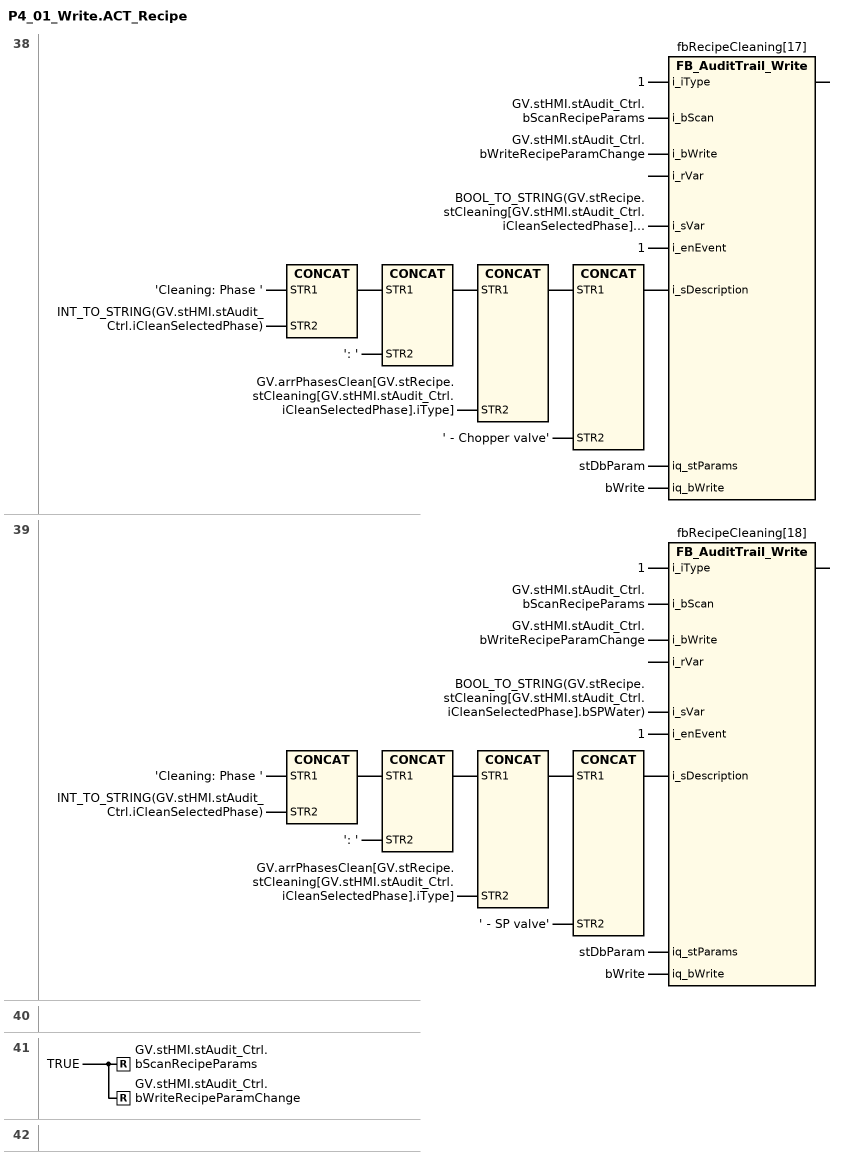
// NETWORK 38
fbRecipeCleaning[17](
    i_iType := 1,
    i_bScan := GV.stHMI.stAudit_Ctrl.bScanRecipeParams,
    i_bWrite := GV.stHMI.stAudit_Ctrl.bWriteRecipeParamChange,
    i_sVar := BOOL_TO_STRING(GV.stRecipe.stCleaning[GV.stHMI.stAudit_Ctrl.iCleanSelectedPhase].bChopperWater),
    i_enEvent := 1,
    i_sDescription := CONCAT(STR1 := CONCAT(STR1 := CONCAT(STR1 := CONCAT(STR1 := 'Cleaning: Phase ', STR2 := INT_TO_STRING(GV.stHMI.stAudit_Ctrl.iCleanSelectedPhase)), STR2 := ': '), STR2 := GV.arrPhasesClean[GV.stRecipe.stCleaning[GV.stHMI.stAudit_Ctrl.iCleanSelectedPhase].iType]), STR2 := ' - Chopper valve'),
    iq_stParams := stDbParam,
    iq_bWrite := bWrite); // FB_AuditTrail_Write

// NETWORK 39
fbRecipeCleaning[18](
    i_iType := 1,
    i_bScan := GV.stHMI.stAudit_Ctrl.bScanRecipeParams,
    i_bWrite := GV.stHMI.stAudit_Ctrl.bWriteRecipeParamChange,
    i_sVar := BOOL_TO_STRING(GV.stRecipe.stCleaning[GV.stHMI.stAudit_Ctrl.iCleanSelectedPhase].bSPWater),
    i_enEvent := 1,
    i_sDescription := CONCAT(STR1 := CONCAT(STR1 := CONCAT(STR1 := CONCAT(STR1 := 'Cleaning: Phase ', STR2 := INT_TO_STRING(GV.stHMI.stAudit_Ctrl.iCleanSelectedPhase)), STR2 := ': '), STR2 := GV.arrPhasesClean[GV.stRecipe.stCleaning[GV.stHMI.stAudit_Ctrl.iCleanSelectedPhase].iType]), STR2 := ' - SP valve'),
    iq_stParams := stDbParam,
    iq_bWrite := bWrite); // FB_AuditTrail_Write

// NETWORK 40

// NETWORK 41
GV.stHMI.stAudit_Ctrl.bScanRecipeParams R= TRUE;
GV.stHMI.stAudit_Ctrl.bWriteRecipeParamChange R= TRUE;

// NETWORK 42
END_ACTION

ACTION ACT_SP:
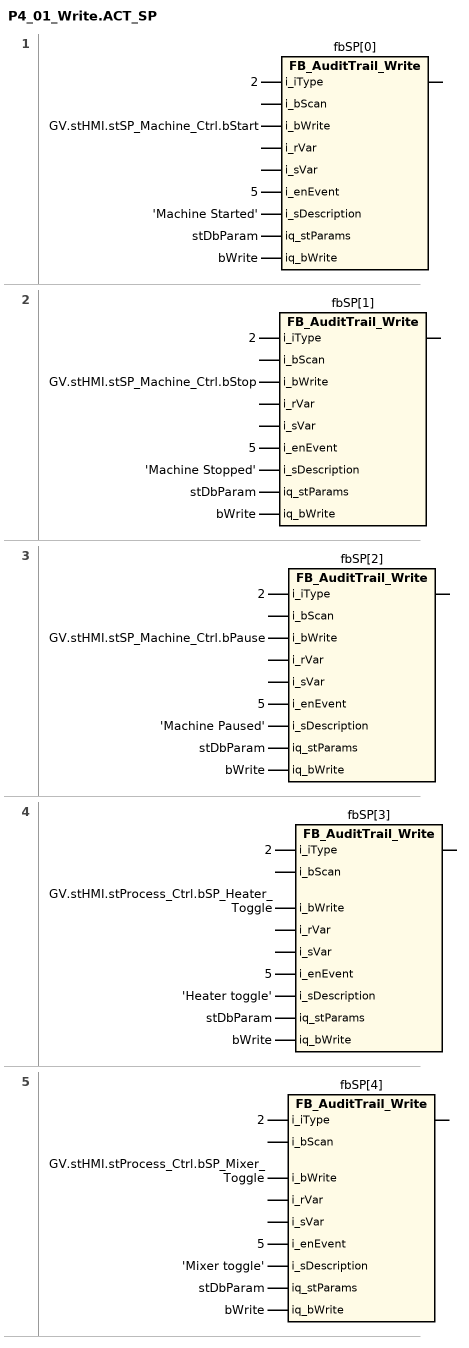
// NETWORK 1
fbSP[0](
    i_iType := 2,
    i_bWrite := GV.stHMI.stSP_Machine_Ctrl.bStart,
    i_enEvent := 5,
    i_sDescription := 'Machine Started',
    iq_stParams := stDbParam,
    iq_bWrite := bWrite); // FB_AuditTrail_Write

// NETWORK 2
fbSP[1](
    i_iType := 2,
    i_bWrite := GV.stHMI.stSP_Machine_Ctrl.bStop,
    i_enEvent := 5,
    i_sDescription := 'Machine Stopped',
    iq_stParams := stDbParam,
    iq_bWrite := bWrite); // FB_AuditTrail_Write

// NETWORK 3
fbSP[2](
    i_iType := 2,
    i_bWrite := GV.stHMI.stSP_Machine_Ctrl.bPause,
    i_enEvent := 5,
    i_sDescription := 'Machine Paused',
    iq_stParams := stDbParam,
    iq_bWrite := bWrite); // FB_AuditTrail_Write

// NETWORK 4
fbSP[3](
    i_iType := 2,
    i_bWrite := GV.stHMI.stProcess_Ctrl.bSP_Heater_Toggle,
    i_enEvent := 5,
    i_sDescription := 'Heater toggle',
    iq_stParams := stDbParam,
    iq_bWrite := bWrite); // FB_AuditTrail_Write

// NETWORK 5
fbSP[4](
    i_iType := 2,
    i_bWrite := GV.stHMI.stProcess_Ctrl.bSP_Mixer_Toggle,
    i_enEvent := 5,
    i_sDescription := 'Mixer toggle',
    iq_stParams := stDbParam,
    iq_bWrite := bWrite); // FB_AuditTrail_Write

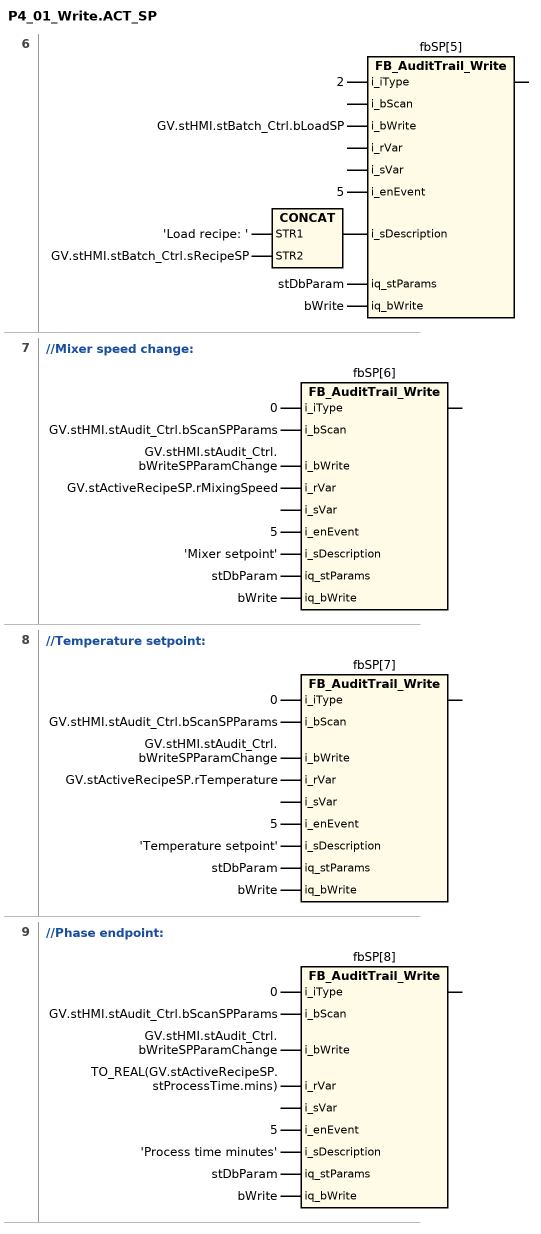
// NETWORK 6
fbSP[5](
    i_iType := 2,
    i_bWrite := GV.stHMI.stBatch_Ctrl.bLoadSP,
    i_enEvent := 5,
    i_sDescription := CONCAT(STR1 := 'Load recipe: ', STR2 := GV.stHMI.stBatch_Ctrl.sRecipeSP),
    iq_stParams := stDbParam,
    iq_bWrite := bWrite); // FB_AuditTrail_Write

// NETWORK 7
// label: //Mixer speed change
fbSP[6](
    i_iType := 0,
    i_bScan := GV.stHMI.stAudit_Ctrl.bScanSPParams,
    i_bWrite := GV.stHMI.stAudit_Ctrl.bWriteSPParamChange,
    i_rVar := GV.stActiveRecipeSP.rMixingSpeed,
    i_enEvent := 5,
    i_sDescription := 'Mixer setpoint',
    iq_stParams := stDbParam,
    iq_bWrite := bWrite); // FB_AuditTrail_Write

// NETWORK 8
// label: //Temperature setpoint
fbSP[7](
    i_iType := 0,
    i_bScan := GV.stHMI.stAudit_Ctrl.bScanSPParams,
    i_bWrite := GV.stHMI.stAudit_Ctrl.bWriteSPParamChange,
    i_rVar := GV.stActiveRecipeSP.rTemperature,
    i_enEvent := 5,
    i_sDescription := 'Temperature setpoint',
    iq_stParams := stDbParam,
    iq_bWrite := bWrite); // FB_AuditTrail_Write

// NETWORK 9
// label: //Phase endpoint
fbSP[8](
    i_iType := 0,
    i_bScan := GV.stHMI.stAudit_Ctrl.bScanSPParams,
    i_bWrite := GV.stHMI.stAudit_Ctrl.bWriteSPParamChange,
    i_rVar := TO_REAL(GV.stActiveRecipeSP.stProcessTime.mins),
    i_enEvent := 5,
    i_sDescription := 'Process time minutes',
    iq_stParams := stDbParam,
    iq_bWrite := bWrite); // FB_AuditTrail_Write

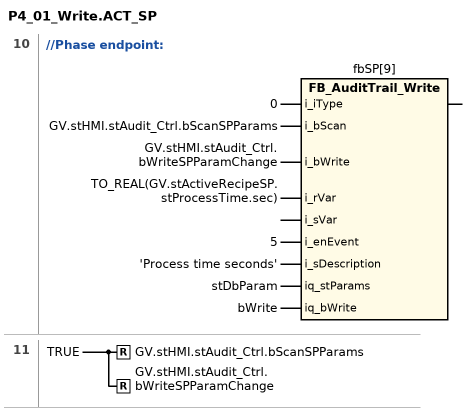
// NETWORK 10
// label: //Phase endpoint
fbSP[9](
    i_iType := 0,
    i_bScan := GV.stHMI.stAudit_Ctrl.bScanSPParams,
    i_bWrite := GV.stHMI.stAudit_Ctrl.bWriteSPParamChange,
    i_rVar := TO_REAL(GV.stActiveRecipeSP.stProcessTime.sec),
    i_enEvent := 5,
    i_sDescription := 'Process time seconds',
    iq_stParams := stDbParam,
    iq_bWrite := bWrite); // FB_AuditTrail_Write

// NETWORK 11
GV.stHMI.stAudit_Ctrl.bScanSPParams R= TRUE;
GV.stHMI.stAudit_Ctrl.bWriteSPParamChange R= TRUE;
END_ACTION

END_PROGRAM

(* stored: Version 1.1.0.1, ProductVersion 3.1.4024.12
   POU P4_01_Write: Id {7d6a380c-9e73-4b04-a35c-8f496aab0134}, SpecialFunc None
   Action ACT_Batch: Id {792cea89-ea65-4751-b10e-b7db5e98c563}
   Action ACT_General: Id {7a1ceb8d-2061-40c7-acaf-dd84c69fb852}
   Action ACT_Recipe: Id {57f0929d-60b6-41a7-acac-3196a0fc3ab7}
   Action ACT_SP: Id {310ecff8-2d2a-402b-b5b9-bea1c2ab6da2} *)
